// TIA Portal V20 export
// export: Created 2025-12-01T14:57:21.7314449Z, ExportSetting None, DisplayName Totally Integrated Automation Portal, DisplayVersion V20 Update 3, DisplayName TIA Portal Openness, DisplayVersion V20 Update 3, DisplayName TIA Portal Version Control Interface, DisplayVersion V20 Update 3, DisplayName STEP 7 Professional, DisplayVersion V20 Update 3, DisplayName STEP 7 Safety, DisplayVersion V20 Update 2, DisplayName WinCC Basic/Comfort/Advanced, DisplayVersion V20 Update 3, DisplayName WinCC Professional, DisplayVersion V20 Update 3, DisplayName WinCC Unified, DisplayVersion V20 Update 3
DATA_BLOCK "DB3000_BYPASS_SAFETY"   // DB3000, F_DB
{ S7_Optimized_Access := 'TRUE' }
// stored: AutoNumber false
   VAR
      Bypass_SF_xxxx_EM : Bool;
      Bypass_SF_xxxx_EM_1 : Bool;
      Bypass_SF_xxxx_EM_2 : Bool;
      Bypass_SF_xxxx_EM_3 : Bool;
      Bypass_SF_xxxx_EM_4 : Bool;
      Bypass_SF_xxxx_EM_5 : Bool;
      Bypass_SF_xxxx_EM_6 : Bool;
      Bypass_SF_xxxx_EM_7 : Bool;
      Bypass_SF_xxxx_EM_8 : Bool;
      Bypass_SF_xxxx_EM_9 : Bool;
      Bypass_SF_xxxx_EM_10 : Bool;
      Bypass_BF_xxBARxx : Bool;
      Bypass_BF_xxBARxx_1 : Bool;
      Bypass_BF_xxBARxx_2 : Bool;
      Bypass_BF_xxBARxx_3 : Bool;
      Bypass_BF_xxBARxx_4 : Bool;
      Bypass_BF_xxBARxx_5 : Bool;
      Bypass_BF_xxBARxx_6 : Bool;
      Bypass_SP_xxxxxx : Bool;
      Bypass_SP_xxxxxx_1 : Bool;
      Bypass_SP_xxxxxx_2 : Bool;
      Bypass_SP_xxxxxx_3 : Bool;
      Bypass_SP_xxxxxx_4 : Bool;
      Bypass_SP_xxxxxx_5 : Bool;
      Bypass_SP_xxxxxx_6 : Bool;
      Bypass_SP_xxxxxx_7 : Bool;
      Bypass_SP_xxxxxx_8 : Bool;
      Bypass_SP_xxxxxx_9 : Bool;
      Bypass_SP_xxxxxx_10 : Bool;
      Bypass_SP_xxxxxx_11 : Bool;
   END_VAR
BEGIN
END_DATA_BLOCK
